// TIA Portal project "FactoryIO_Template_S7-1500_V15_V16" (V16)

(* hardware
DEVICE "S71500/ET200MP-Station_1"  S7-1500 station
   slot 0: "Profilschiene_0"  Rack  6ES7 590-1***0-0AA0
   slot 1: "PLC_1"  CPU 1512C-1 PN  6ES7 512-1CK01-0AB0  V2.8
      slot 3: "CPU-Display_1"  6ES7591-1AA00-0AA0
      slot 32768: "PROFINET-Schnittstelle_1"  X1
         slot 32769: "Port_1"  X1 P1
         slot 32770: "Port_2"  X1 P2
      slot 34817: "Virtual CP interface port_1"  Virtual CP interface port  Virtual CP interface port
   slot 2: "AI 8xU/I/RTD/TC ST_1"  AI 8xU/I/RTD/TC ST  6ES7 531-7KF00-0AB0  V2.0
   slot 3: "AI 8xU/I/RTD/TC ST_2"  AI 8xU/I/RTD/TC ST  6ES7 531-7KF00-0AB0  V2.0
   slot 4: "AI 8xU/I/RTD/TC ST_3"  AI 8xU/I/RTD/TC ST  6ES7 531-7KF00-0AB0  V2.0
   slot 5: "AI 8xU/I/RTD/TC ST_4"  AI 8xU/I/RTD/TC ST  6ES7 531-7KF00-0AB0  V2.0
   slot 6: "DI 16x24VDC BA_1"  DI 16x24VDC BA  6ES7 521-1BH10-0AA0  V1.0
DEVICE "HMI_2"  KTP700 Basic PN
   slot 0: "HMI_2"  KTP700 Basic PN  6AV2 123-2GB03-0AX0  16.0.0.0
   slot 1: "HMI_RT_2"  KTP700 Basic PN  6AV2 123-2GB03-0AX0  16.0.0.0
   slot 5: "HMI_2.IE_CP_1"  PROFINET Interface  16.0.0.0
      slot 1: "PROFINET Interface_1"  PROFINET Interface
         slot 1: "Port_1"  Port
*)

// ===== PLC "PLC_1"  CPU 1512C-1 PN =====

VAR_GLOBAL   // PLC tag table "Standard-Variablentabelle"
   "Tag_1" AT %M0.1 : Bool;
   "Tag_2" AT %M0.0 : Bool;
END_VAR

VAR_GLOBAL   // PLC tag table "Inputs"
   "Flow_Rate_Sensor" AT %I1.0 : Bool;
   "Float_switch_overflow" AT %I1.1 : Bool;   // S111
   "Float_switch_threshold" AT %I1.2 : Bool;   // S112
   "Low_Level_Capacitive_Sensor" AT %I1.3 : Bool;   // B114
   "High_Level_Capacitive_Sensor" AT %I1.4 : Bool;   // B113
   "Micro_switch_valve_closed" AT %I1.5 : Bool;
   "Micro_switch_valve_open" AT %I1.6 : Bool;
   "Ultrasonic_Sensor" AT %IW96 : Int;
END_VAR

VAR_GLOBAL   // PLC tag table "Outputs"
   "Solenoid_on/off" AT %Q1.0 : Bool;
   "Heater_on/off" AT %Q1.1 : Bool;
   "Relay KF1_Pump mode" AT %Q1.2 : Bool;
   "Pump_on/off" AT %Q1.3 : Bool;
   "KF6_Proportional valve" AT %Q1.4 : Bool;
   "KF2_Fan" AT %Q1.5 : Bool;
   "Pump_P101" AT %QW96 : Int;
END_VAR

VAR_GLOBAL   // PLC tag table "Factory tags"
   "FactoryIO_running" AT %I0.3 : Bool;
   "Ultrasonic_Sensor_factory" AT %ID30 : Real;
   "Fill valve" AT %QD30 : Real;
   "Discharge valve" AT %QD34 : Real;
   "SP" AT %QD38 : DInt;
   "Flow meter" AT %ID34 : Real;
   "setpoint" AT %ID38 : Real;
   "PV" AT %QD42 : DInt;
   "Start" AT %I0.0 : Bool;
   "Reset" AT %I0.1 : Bool;
   "Stop" AT %I0.2 : Bool;
   "Start light" AT %Q0.0 : Bool;
   "Reset light" AT %Q0.1 : Bool;
   "Stop light" AT %Q0.2 : Bool;
END_VAR

// folder: Sys_par

DATA_BLOCK "sys_utils"   // DB3
{ S7_Optimized_Access := 'TRUE' }
VERSION : 0.1
   VAR
      "toggle tags" : Bool;
      process_type : Int := 0;
      _xState_pump : Bool;
      _xState_discharge : Bool;
      _xState_Start : Bool;
      _xState_Reset : Bool;
      _xState_Stop : Bool;
      _xState_PIDState : Bool;
   END_VAR
BEGIN
END_DATA_BLOCK

DATA_BLOCK "parameters"   // DB4
{ S7_Optimized_Access := 'TRUE' }
VERSION : 0.1
   VAR
      "Process Value" : Real;
      setpoint : DInt := 0;
      setpoint_pid : Real;
      flowrate : Real;
      ModeActivate : Bool;
      ManualEnable : Bool;
      InactiveEnable : Bool;
      ManualValue : Real := 80.0;
      Inactive : Int := 0;
      Reset : Bool;
      "Error_Discharge valve" : Real;
      "Flow_Meter buffer" : Real;
      "Level Buffer" : Real;
      "Setpoint buffer" : Real;
      Error : Real;
      PWM_DISABLE : Bool;
   END_VAR
BEGIN
END_DATA_BLOCK

// folder: (top level)

FUNCTION "Control_Unit" : Void   // FC1, LAD
{ S7_Optimized_Access := 'TRUE' }
VERSION : 0.1
   VAR_TEMP
      stop_light : Bool;
      start_light : Bool;
   END_VAR
   VAR_TEMP   // added for the SCL form of the ladder/FBD networks
      _w1 : Bool;
      _w2 : Bool;
   END_VAR
BEGIN

REGION Network 1: Stop condition
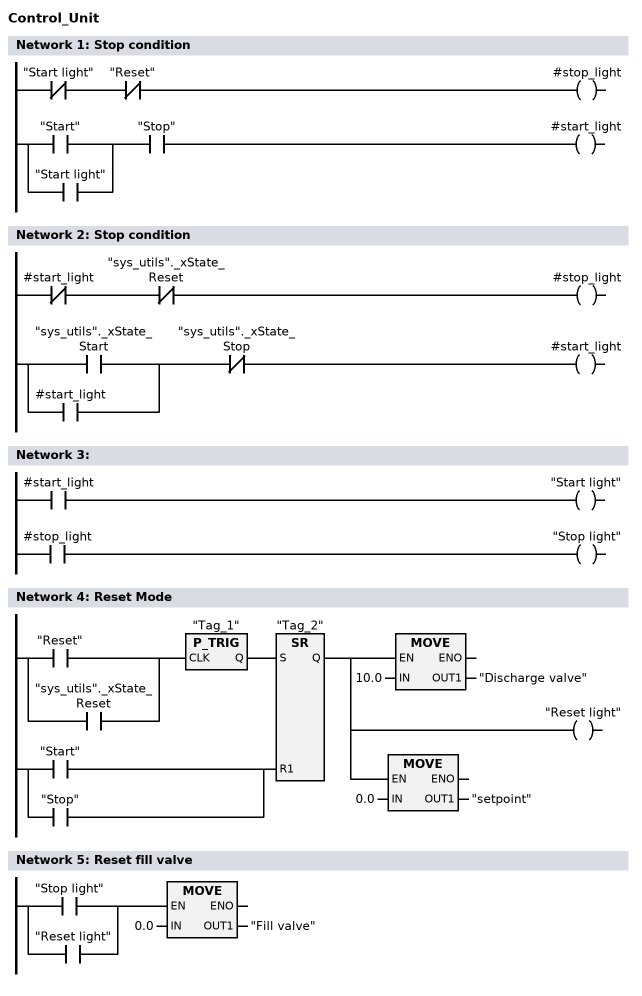
   RUNG wire#powerrail
      I_Contact( "Start light" )
      I_Contact( "Reset" )
      Coil( #stop_light )
   END_RUNG
   RUNG wire#powerrail
      Contact( "Start" )
      wire#w1
      Contact( "Stop" )
      Coil( #start_light )
   END_RUNG
   RUNG wire#powerrail
      Contact( "Start light" )
   END_RUNG wire#w1
   // the same network as SCL:
   #stop_light := NOT "Start light" AND NOT "Reset";
   #start_light := ("Start" OR "Start light") AND "Stop";
END_REGION

REGION Network 2: Stop condition
   RUNG wire#powerrail
      I_Contact( #start_light )
      I_Contact( "sys_utils"._xState_Reset )
      Coil( #stop_light )
   END_RUNG
   RUNG wire#powerrail
      Contact( "sys_utils"._xState_Start )
      wire#w1
      I_Contact( "sys_utils"._xState_Stop )
      Coil( #start_light )
   END_RUNG
   RUNG wire#powerrail
      Contact( #start_light )
   END_RUNG wire#w1
   // the same network as SCL:
   #stop_light := NOT #start_light AND NOT "sys_utils"._xState_Reset;
   #start_light := ("sys_utils"._xState_Start OR #start_light) AND NOT "sys_utils"._xState_Stop;
END_REGION

REGION Network 3
   RUNG wire#powerrail
      Contact( #start_light )
      Coil( "Start light" )
   END_RUNG
   RUNG wire#powerrail
      Contact( #stop_light )
      Coil( "Stop light" )
   END_RUNG
   // the same network as SCL:
   "Start light" := #start_light;
   "Stop light" := #stop_light;
END_REGION

REGION Network 4: Reset Mode
   RUNG wire#powerrail
      Contact( "Reset" )
      wire#w1
      P_Trig( "Tag_1" )
      S_SR(operand := "Tag_2", r1 := wire#w2)
      wire#w3
      Move(in := 10.0, out1 => "Discharge valve")
   END_RUNG
   RUNG wire#powerrail
      Contact( "sys_utils"._xState_Reset )
   END_RUNG wire#w1
   RUNG wire#powerrail
      Contact( "Start" )
   END_RUNG wire#w2
   RUNG wire#powerrail
      Contact( "Stop" )
   END_RUNG wire#w2
   RUNG wire#w3
      Coil( "Reset light" )
   END_RUNG
   RUNG wire#w3
      Move(in := 0.0, out1 => "setpoint")
   END_RUNG
   // the same network as SCL:
   #_w1 := "Reset" OR "sys_utils"._xState_Reset;
   #_w2 := #_w1 AND NOT "Tag_1";   // rising edge
   "Tag_1" := #_w1;
   IF #_w2 THEN
       "Tag_2" := TRUE;   // SR flip-flop
   END_IF;
   IF "Start" OR "Stop" THEN "Tag_2" := FALSE; END_IF;
   IF "Tag_2" THEN "Discharge valve" := 10.0; END_IF;
   "Reset light" := "Tag_2";
   IF "Tag_2" THEN "setpoint" := 0.0; END_IF;
END_REGION

REGION Network 5: Reset fill valve
   RUNG wire#powerrail
      Contact( "Stop light" )
      wire#w1
      Move(in := 0.0, out1 => "Fill valve")
   END_RUNG
   RUNG wire#powerrail
      Contact( "Reset light" )
   END_RUNG wire#w1
   // the same network as SCL:
   IF "Stop light" OR "Reset light" THEN "Fill valve" := 0.0; END_IF;
END_REGION
END_FUNCTION

FUNCTION "height_conversion" : Void   // FC3, LAD
{ S7_Optimized_Access := 'TRUE' }
VERSION : 0.1
   VAR_INPUT
      height_sensor : Real;
   END_VAR
   VAR_OUTPUT
      scaled_height : DInt;
   END_VAR
   VAR_TEMP
      norm_height : Real;
   END_VAR
BEGIN

REGION Network 1: Height Conversion
   // 1. Normalize the sensor output data between 0.0 and 1.0
   // 2. Scale the normalized data between minimum and maximum scale reading
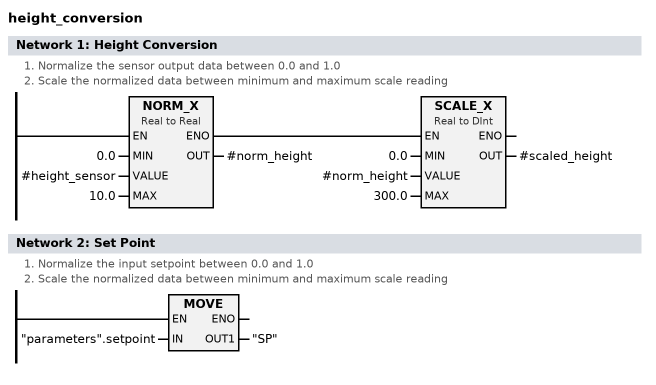
   RUNG wire#powerrail
      { S7_Templates := "[SrcType := Real, DestType := Real]" } Normalize(min := 0.0, value := #height_sensor, max := 10.0, out => #norm_height)
      { S7_Templates := "[SrcType := Real, DestType := DInt]" } Scale(min := 0.0, value := #norm_height, max := 300.0, out => #scaled_height)
   END_RUNG
   // the same network as SCL:
   #norm_height := NORM_X(MIN := 0.0, VALUE := #height_sensor, MAX := 10.0);
   #scaled_height := SCALE_X(MIN := 0.0, VALUE := #norm_height, MAX := 300.0);
END_REGION

REGION Network 2: Set Point
   // 1. Normalize the input setpoint between 0.0 and 1.0
   // 2. Scale the normalized data between minimum and maximum scale reading
   RUNG wire#powerrail
      Move(in := "parameters".setpoint, out1 => "SP")
   END_RUNG
   // the same network as SCL:
   "SP" := "parameters".setpoint;
END_REGION
END_FUNCTION

FUNCTION "MHJ-PLC-Lab-Function-S71500" : Void   // FC9000, SCL
{ S7_Optimized_Access := 'TRUE' }
VERSION : 0.1
   VAR_TEMP
      Value : Byte;
      ForCounter : Int;
   END_VAR
   VAR CONSTANT
      Value_01_DW : DWord := 16#1223_5486;
      Value_02_DW : DWord := 16#A6C9_D1F5;
   END_VAR
BEGIN

   #Value:=PEEK(area := 16#82,
        dbNumber := 0,
        byteOffset := 511);
   #Value := #Value + 1;

   POKE(area := 16#82,
        dbNumber := 0,
        byteOffset := 511,
        value := #Value);

   POKE(area := 16#82,
        dbNumber := 0,
        byteOffset := 1016,
        value := #Value_01_DW);
   POKE(area := 16#82,
        dbNumber := 0,
        byteOffset := 1020,
        value := #Value_02_DW);

   FOR #ForCounter := 0 TO 63 DO
       #Value:=PEEK(area := 16#1,
            dbNumber := 0,
            byteOffset := #ForCounter);
       POKE(area := 16#81,
            dbNumber := 0,
            byteOffset := #ForCounter,
            value := #Value);
   END_FOR;
   #Value := PEEK(area := 16#1,
                  dbNumber := 0,
                  byteOffset := 512);
   POKE(area := 16#82,
        dbNumber := 0,
        byteOffset := 512,
        value := #Value);
END_FUNCTION

ORGANIZATION_BLOCK "Main"   // OB1, LAD, ProgramCycle
TITLE = "Main Program Sweep (Cycle)"
{ S7_Optimized_Access := 'TRUE' }
VERSION : 0.1
   VAR_INPUT
      Initial_Call : Bool;   // Initial call of this OB
      Remanence : Bool;   // =True, if remanent data are available
   END_VAR
BEGIN

REGION Network 1
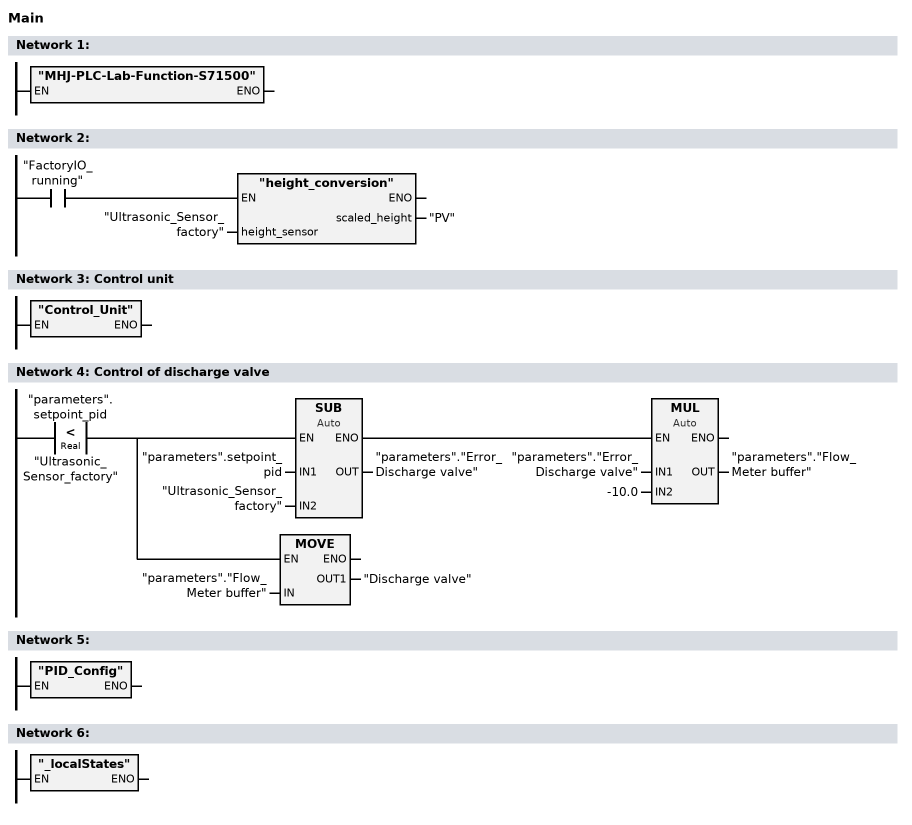
   RUNG wire#powerrail
      "MHJ-PLC-Lab-Function-S71500"()
   END_RUNG
   // the same network as SCL:
   "MHJ-PLC-Lab-Function-S71500"();
END_REGION

REGION Network 2
   RUNG wire#powerrail
      Contact( "FactoryIO_running" )
      "height_conversion"(height_sensor := "Ultrasonic_Sensor_factory", scaled_height => "PV")
   END_RUNG
   // the same network as SCL:
   IF "FactoryIO_running" THEN
       "height_conversion"(height_sensor := "Ultrasonic_Sensor_factory", scaled_height => "PV");
   END_IF;
END_REGION

REGION Network 3: Control unit
   RUNG wire#powerrail
      "Control_Unit"()
   END_RUNG
   // the same network as SCL:
   "Control_Unit"();
END_REGION

REGION Network 4: Control of discharge valve
   RUNG wire#powerrail
      { S7_Templates := "SrcType := Real" } LT_Contact(in1 := "parameters".setpoint_pid, in2 := "Ultrasonic_Sensor_factory")
      wire#w1
      Sub(in1 := "parameters".setpoint_pid, in2 := "Ultrasonic_Sensor_factory", out => "parameters"."Error_Discharge valve")
      Mul(in1 := "parameters"."Error_Discharge valve", in2 := -10.0, out => "parameters"."Flow_Meter buffer")
   END_RUNG
   RUNG wire#w1
      Move(in := "parameters"."Flow_Meter buffer", out1 => "Discharge valve")
   END_RUNG
   // the same network as SCL:
   IF "parameters".setpoint_pid < "Ultrasonic_Sensor_factory" THEN
       "parameters"."Error_Discharge valve" := "parameters".setpoint_pid - "Ultrasonic_Sensor_factory";
       "parameters"."Flow_Meter buffer" := "parameters"."Error_Discharge valve" * (-10.0);
       "Discharge valve" := "parameters"."Flow_Meter buffer";
   END_IF;
END_REGION

REGION Network 5
   RUNG wire#powerrail
      "PID_Config"()
   END_RUNG
   // the same network as SCL:
   "PID_Config"();
END_REGION

REGION Network 6
   RUNG wire#powerrail
      "_localStates"()
   END_RUNG
   // the same network as SCL:
   "_localStates"();
END_REGION
END_ORGANIZATION_BLOCK

ORGANIZATION_BLOCK "Cyclic interrupt PID"   // OB30, LAD, CyclicInterrupt
{ S7_Optimized_Access := 'TRUE' }
VERSION : 0.1
   VAR_INPUT
      Initial_Call : Bool;   // Initial call of this OB
      Event_Count : Int;   // Events discarded
   END_VAR
BEGIN

REGION Network 1
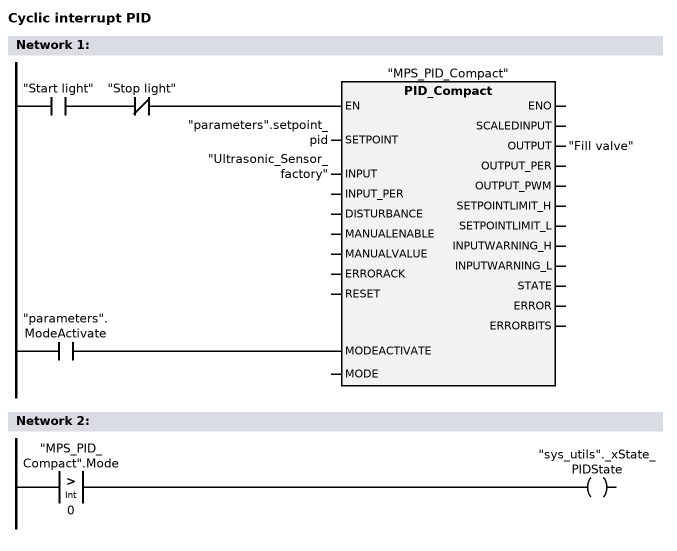
   IF "Start light" AND NOT "Stop light" THEN
       "MPS_PID_Compact"(Setpoint := "parameters".setpoint_pid,   // PID_Compact
                         Input := "Ultrasonic_Sensor_factory",
                         ModeActivate := "parameters".ModeActivate,
                         Output => "Fill valve");
   END_IF;
END_REGION

REGION Network 2
   RUNG wire#powerrail
      { S7_Templates := "SrcType := Int" } GT_Contact(in1 := "MPS_PID_Compact".Mode, in2 := 0)
      Coil( "sys_utils"._xState_PIDState )
   END_RUNG
   // the same network as SCL:
   "sys_utils"._xState_PIDState := "MPS_PID_Compact".Mode > 0;
END_REGION
END_ORGANIZATION_BLOCK

// folder: Sys_par

FUNCTION "PID_Config" : Void   // FC2, LAD
{ S7_Optimized_Access := 'TRUE' }
VERSION : 0.1
   VAR_TEMP
      norm_setpoint : Real;
   END_VAR
BEGIN

REGION Network 1: enable mode
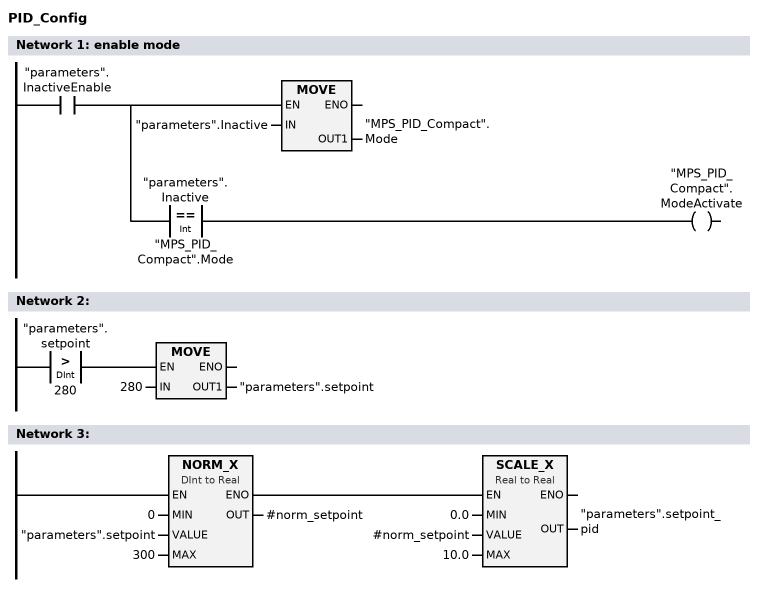
   RUNG wire#powerrail
      Contact( "parameters".InactiveEnable )
      wire#w1
      Move(in := "parameters".Inactive, out1 => "MPS_PID_Compact".Mode)
   END_RUNG
   RUNG wire#w1
      { S7_Templates := "SrcType := Int" } EQ_Contact(in1 := "parameters".Inactive, in2 := "MPS_PID_Compact".Mode)
      Coil( "MPS_PID_Compact".ModeActivate )
   END_RUNG
   // the same network as SCL:
   IF "parameters".InactiveEnable THEN "MPS_PID_Compact".Mode := "parameters".Inactive; END_IF;
   "MPS_PID_Compact".ModeActivate := "parameters".InactiveEnable AND ("parameters".Inactive = "MPS_PID_Compact".Mode);
END_REGION

REGION Network 2
   RUNG wire#powerrail
      { S7_Templates := "SrcType := DInt" } GT_Contact(in1 := "parameters".setpoint, in2 := 280)
      Move(in := 280, out1 => "parameters".setpoint)
   END_RUNG
   // the same network as SCL:
   IF "parameters".setpoint > 280 THEN "parameters".setpoint := 280; END_IF;
END_REGION

REGION Network 3
   RUNG wire#powerrail
      { S7_Templates := "[SrcType := DInt, DestType := Real]" } Normalize(min := 0, value := "parameters".setpoint, max := 300, out => #norm_setpoint)
      { S7_Templates := "[SrcType := Real, DestType := Real]" } Scale(min := 0.0, value := #norm_setpoint, max := 10.0, out => "parameters".setpoint_pid)
   END_RUNG
   // the same network as SCL:
   #norm_setpoint := NORM_X(MIN := 0, VALUE := "parameters".setpoint, MAX := 300);
   "parameters".setpoint_pid := SCALE_X(MIN := 0.0, VALUE := #norm_setpoint, MAX := 10.0);
END_REGION
END_FUNCTION

FUNCTION "_localStates" : Void   // FC4, LAD
{ S7_Optimized_Access := 'TRUE' }
VERSION : 0.1
BEGIN

REGION Network 1: Pump state
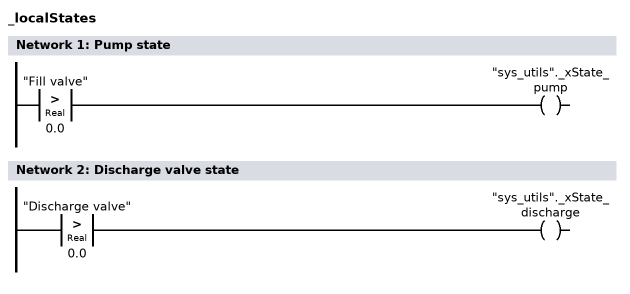
   RUNG wire#powerrail
      { S7_Templates := "SrcType := Real" } GT_Contact(in1 := "Fill valve", in2 := 0.0)
      Coil( "sys_utils"._xState_pump )
   END_RUNG
   // the same network as SCL:
   "sys_utils"._xState_pump := "Fill valve" > 0.0;
END_REGION

REGION Network 2: Discharge valve state
   RUNG wire#powerrail
      { S7_Templates := "SrcType := Real" } GT_Contact(in1 := "Discharge valve", in2 := 0.0)
      Coil( "sys_utils"._xState_discharge )
   END_RUNG
   // the same network as SCL:
   "sys_utils"._xState_discharge := "Discharge valve" > 0.0;
END_REGION
END_FUNCTION

(* ===== HMI "HMI_RT_2" =====
system functions are stored by id; their names below are inferred from use
connection "HMI_Connection_2": ETHERNET, SMART_S7_1500_OMS

HMI tags "Default tag table"
   "Tag_ScreenNumber" : UInt, internal
   "PV" : DInt = PLC PV AT %QD42, 1 s
   "SP" : DInt = PLC SP AT %QD38, 1 s
   "MPS_PID_Compact_CtrlParamsBackUp_Gain" : Real = PLC MPS_PID_Compact.CtrlParamsBackUp.Gain, 1 s
   "MPS_PID_Compact_CtrlParamsBackUp_Ti" : Real = PLC MPS_PID_Compact.CtrlParamsBackUp.Ti, 1 s
   "MPS_PID_Compact_CtrlParamsBackUp_Td" : Real = PLC MPS_PID_Compact.CtrlParamsBackUp.Td, 1 s
   "setpoint" : Real = PLC setpoint AT %ID38, 1 s
   "Start" : Bool = PLC Start AT %I0.0, 1 s
   "Start light" : Bool = PLC "Start light" AT %Q0.0, 1 s
   "Stop" : Bool = PLC Stop AT %I0.2, 1 s
   "Stop light" : Bool = PLC "Stop light" AT %Q0.2, 1 s
   "MPS_PID_Compact_Mode" : Int = PLC MPS_PID_Compact.Mode, 1 s
   "MPS_PID_Compact_ModeActivate" : Bool = PLC MPS_PID_Compact.ModeActivate, 1 s
   "parameters_InactiveEnable" : Bool = PLC parameters.InactiveEnable, 1 s
   "parameters_setpoint" : DInt = PLC parameters.setpoint, 1 s
   "sys_utils_toggle tags" : Bool = PLC sys_utils."toggle tags", 1 s
   "Reset" : Bool = PLC Reset AT %I0.1, 1 s
   "Reset light" : Bool = PLC "Reset light" AT %Q0.1, 1 s
   "sys_utils_process_type" : Int = PLC sys_utils.process_type, 1 s
   "sys_utils__xState_discharge" : Bool = PLC sys_utils._xState_discharge, 1 s
   "sys_utils__xState_pump" : Bool = PLC sys_utils._xState_pump, 1 s
   "sys_utils__xState_Start" : Bool = PLC sys_utils._xState_Start, 1 s
   "sys_utils__xState_Stop" : Bool = PLC sys_utils._xState_Stop, 1 s
   "parameters_ModeActivate" : Bool = PLC parameters.ModeActivate, 1 s
   "sys_utils__xState_Reset" : Bool = PLC sys_utils._xState_Reset, 1 s
   "sys_utils__xState_PIDState" : Bool = PLC sys_utils._xState_PIDState, 1 s

HMI tags "Local Template"
   "_iScreenNumber" : Int, internal
   "_xState_Btn_Overview" : Bool, internal
   "_xState_Btn_Alarm" : Bool, internal
   "_xState_Btn_Recipe" : Bool, internal
   "_xState_Btn_Settings" : Bool, internal
   "_xState_Btn_Level_Overview" : Bool, internal
   "_xState_Btn_Level_Config" : Bool, internal
   "_xState_Btn_Alarm_Buffer" : Bool, internal
   "_xState_Btn_ToggleTags" : Bool, internal
   "_sUserName" : WString[254], internal
   "_iUserGroupNumber" : Int, internal

text list "Text_list_Modes": 3 'Automatic'; 4 'Manual'

text list "Text_list_ToggleTags": 0 'Tags'; 1 'Name'

text list "Text_list_ProcessNames": 1 'Level Control'; 2 'Flow Control'; 3 'Temperature'; 4 'Pressure'; 0 'Home'

graphic list "GraphList_Btn_Template_Settings": 0 'Graphic_13'; 1 'Graphic_12'

graphic list "GraphList_Proportional_Valve": 0 'Graphic_45'; 1 'Graphic_46'

graphic list "GraphList_Pump": 0 'Graphic_27'; 1 'Graphic_26'

graphic list "GraphList_Btn_Template_Recipe": 0 'Graphic_14'; 1 'Graphic_15'

graphic list "GraphList_Btn_Template_Alarm": 0 'Graphic_16'; 1 'Graphic_17'

graphic list "GraphList_Btn_Template_Overview": 0 'Graphic_19'; 1 'Graphic_18'

screen "Alarm" 800x480, template "Template_overview"
   on GenerateScreen: SetBit("_xState_Btn_Alarm"); SetTag("_iScreenNumber", 10)
   on ClearScreen: ResetBit("_xState_Btn_Alarm")
   AlarmView "Alarm view_1" at 5,48 size 592x422
   Button "Template_Button_4" at 600,409 size 83x58; TextOff 'Text'; PictureList "GraphList_Btn_Template_Settings"; PictureOff "Graphic_49"; PictureOn "Graphic_50"; Authorization "Operation"
      ProcessValue <- "_xState_Btn_Settings"
   Button "Template_Button_1" at 600,48 size 83x58; TextOff 'Text'; PictureList "GraphList_Btn_Template_Settings"; PictureOff "Graphic_54"; PictureOn "Graphic_50"
      on Release: ActivateScreen("Alarm Buffer", 0)
      ProcessValue <- "_xState_Btn_Settings"

screen "Level Config" 800x480, template "Template"
   on GenerateScreen: SetBit("_xState_Btn_Level_Config"); SetTag("_iScreenNumber", 2)
   on ClearScreen: ResetBit("_xState_Btn_Level_Config")
   TrendView "Trend view_1" at 38,167 size 644x300
   IOField "I/O field_1" at 442,76 size 105x27; FormatPattern 999.99
      ProcessValue <- "MPS_PID_Compact_CtrlParamsBackUp_Gain"
   IOField "I/O field_2" at 442,105 size 105x27; FormatPattern 99.99
      ProcessValue <- "MPS_PID_Compact_CtrlParamsBackUp_Ti"
   IOField "I/O field_3" at 442,135 size 105x27; FormatPattern 99.99
      ProcessValue <- "MPS_PID_Compact_CtrlParamsBackUp_Td"
   TextField "Text field_1" at 553,80 size 107x23; Text 'Proportional'
   TextField "Text field_2" at 552,108 size 71x23; Text 'Integral'
   TextField "Text field_3" at 552,136 size 89x23; Text 'Derivative'
   Button "Button_1" at 442,47 size 218x28; TextOff 'Save PID Parameters'
   Button "Button_2" at 200,53 size 96x30; TextOff 'Enable'
      on Press: SetBit("parameters_ModeActivate")
      on Release: ResetBit("parameters_ModeActivate")
      Appearance <- "sys_utils__xState_PIDState"
   Button "Button_5" at 305,53 size 96x31; TextOff 'Disable'
      on Release: ResetBit("parameters_InactiveEnable")
      on Press: SetBit("parameters_InactiveEnable")
   IOField "I/O field_4" at 43,129 size 105x33; FormatPattern 999
      ProcessValue <- "parameters_setpoint"
   TextField "Text field_4" at 43,106 size 75x23; Text 'SetPoint'
   IOField "I/O field_5" at 278,126 size 105x33; FormatPattern 999
      ProcessValue <- "PV"
   TextField "Text field_5" at 272,105 size 118x23; Text 'Process Value'
   SymbolicIOField "Symbolic I/O field_1" at 38,51 size 159x32; TextOff '0'; TextOn '1'; TextList "Text_list_Modes"
      ProcessValue <- "MPS_PID_Compact_Mode"
   Button "Button_3" at 157,0 size 160x40; TextOff 'OverView'
      Appearance <- "_xState_Btn_Level_Overview"
      on Release: ActivateScreen("Level OverView", 0); SetBit("_xState_Btn_Level_Overview"); ResetBit("_xState_Btn_Level_Config")
   Button "Button_4" at 322,1 size 145x40; TextOff 'Configuration'
      on Release: ActivateScreen("Level Config", 0); SetBit("_xState_Btn_Level_Config"); ResetBit("_xState_Btn_Level_Overview")
      Appearance <- "_xState_Btn_Level_Config"

screen "Level OverView" 800x480, template "Template"
   on GenerateScreen: SetBit("_xState_Btn_Level_Overview"); SetTag("_iScreenNumber", 2)
   on ClearScreen: ResetBit("_xState_Btn_Level_Overview")
   GraphicView "Graphic view_4" at 128,89 size 150x187; Picture "Graphic_25"
   GraphicView "Graphic view_1" at 416,163 size 148x178; Picture "Graphic_25"
   Circle "Circle_5" at 393,433 size 25x25
      Appearance <- "sys_utils__xState_PIDState"
   GraphicView "Graphic view_21" at 319,78 size 45x23; Picture "Graphic_40"
   GraphicView "Graphic view_25" at 222,281 size 40x21; Picture "Graphic_40"
   GraphicView "Graphic view_18" at 85,270 size 31x44; Picture "Graphic_39"
   GraphicView "Graphic view_20" at 502,367 size 51x31; Picture "Graphic_40"
   Bar "Bar_1" at 140,124 size 128x115; MinimumValue 0; MaximumValue 300
      ProcessValue <- "PV"
   Button "Button_3" at 157,0 size 160x40; TextOff 'OverView'
      on Release: ActivateScreen("Level OverView", 0); SetBit("_xState_Btn_Level_Overview"); ResetBit("_xState_Btn_Level_Config")
      Appearance <- "_xState_Btn_Level_Overview"
   Button "Button_4" at 322,1 size 145x40; TextOff 'Configuration'
      on Release: ActivateScreen("Level Config", 0); SetBit("_xState_Btn_Level_Config"); ResetBit("_xState_Btn_Level_Overview")
      Appearance <- "_xState_Btn_Level_Config"
   Button "Button_1" at 432,372 size 43x52; TextOff 'Text'; PictureList "GraphList_Pump"
      ProcessValue <- "sys_utils__xState_pump"
   GraphicView "Graphic view_2" at 116,382 size 322x34; Picture "Graphic_28"
   GraphicView "Graphic view_7" at 81,383 size 36x32; Picture "Graphic_32"
   GraphicView "Graphic view_3" at 83,310 size 34x75; Picture "Graphic_33"
   GraphicView "Graphic view_5" at 111,211 size 30x34; Picture "Graphic_28"
   GraphicView "Graphic view_6" at 474,333 size 34x38; Picture "Graphic_33"
   GraphicView "Graphic view_8" at 474,363 size 35x41; Picture "Graphic_36"
   GraphicView "Graphic view_9" at 191,258 size 34x22; Picture "Graphic_33"
   GraphicView "Graphic view_10" at 259,275 size 173x34; Picture "Graphic_28"
   GraphicView "Graphic view_11" at 266,116 size 27x34; Picture "Graphic_28"
   GraphicView "Graphic view_12" at 357,71 size 137x34; Picture "Graphic_28"
   GraphicView "Graphic view_13" at 524,71 size 83x34; Picture "Graphic_28"
   GraphicView "Graphic view_14" at 547,187 size 59x34; Picture "Graphic_28"
   GraphicView "Graphic view_15" at 604,98 size 34x94; Picture "Graphic_33"
   GraphicView "Graphic view_16" at 194,60 size 31x41; Picture "Graphic_37"
   GraphicView "Graphic view_17" at 190,276 size 36x32; Picture "Graphic_32"
   GraphicView "Graphic view_19" at 290,114 size 37x37; Picture "Graphic_42"
   GraphicView "Graphic view_23" at 291,104 size 34x16; Picture "Graphic_33"
   GraphicView "Graphic view_24" at 292,75 size 33x31; Picture "Graphic_43"
   GraphicView "Graphic view_26" at 84,212 size 33x33; Picture "Graphic_43"
   GraphicView "Graphic view_27" at 83,241 size 34x38; Picture "Graphic_33"
   GraphicView "Graphic view_28" at 544,366 size 30x34; Picture "Graphic_28"
   GraphicView "Graphic view_29" at 602,186 size 37x37; Picture "Graphic_42"
   GraphicView "Graphic view_30" at 603,70 size 37x37; Picture "Graphic_44"
   Button "Button_2" at 491,67 size 36x41; TextOff 'Text'; PictureList "GraphList_Proportional_Valve"
      ProcessValue <- "sys_utils__xState_discharge"
   GraphicView "Graphic view_31" at 560,343 size 82x83; Picture "Graphic_48"
   TextField "Text field_1" at 58,187 size 45x23; Text 'S112'
      Visibility <- "_xState_Btn_ToggleTags"
   TextField "Text field_2" at 224,50 size 46x23; Text 'B102'
      Visibility <- "_xState_Btn_ToggleTags"
   TextField "Text field_3" at 340,186 size 46x23; Text 'B113'
      Visibility <- "_xState_Btn_ToggleTags"
   TextField "Text field_4" at 594,287 size 46x23; Text 'B114'
      Visibility <- "_xState_Btn_ToggleTags"
   TextField "Text field_5" at 424,140 size 45x23; Text 'S111'
      Visibility <- "_xState_Btn_ToggleTags"
   TextField "Text field_6" at 466,48 size 113x20; Text 'Proportion valve'
      Visibility <- "_xState_Btn_ToggleTags"
   TextField "Text field_7" at 120,287 size 46x23; Text 'V101'
      Visibility <- "_xState_Btn_ToggleTags"
   TextField "Text field_8" at 221,302 size 46x23; Text 'V110'
      Visibility <- "_xState_Btn_ToggleTags"
   TextField "Text field_9" at 504,396 size 46x23; Text 'V105'
      Visibility <- "_xState_Btn_ToggleTags"
   TextField "Text field_10" at 319,103 size 46x23; Text 'V112'
      Visibility <- "_xState_Btn_ToggleTags"
   TextField "Text field_11" at 508,142 size 82x20; Text 'Float switch'
      Visibility <- "_xState_Btn_ToggleTags"
   TextField "Text field_12" at 580,266 size 101x20; Text 'Low Level Cap.'
      Visibility <- "_xState_Btn_ToggleTags"
   TextField "Text field_13" at 288,165 size 103x20; Text 'High Level Cap.'
      Visibility <- "_xState_Btn_ToggleTags"
   TextField "Text field_14" at 56,162 size 82x20; Text 'Float switch'
      Visibility <- "_xState_Btn_ToggleTags"
   TextField "Text field_15" at 224,68 size 69x20; Text 'Ultrasonic'
      Visibility <- "_xState_Btn_ToggleTags"
   TextField "Text field_16" at 344,415 size 49x26; Text 'PID'
   SymbolicIOField "Symbolic I/O field_1" at 694,198 size 97x32; TextOff '0'; TextOn '1'; TextList "Text_list_ToggleTags"
      ProcessValue <- "_xState_Btn_ToggleTags"
   TextField "Text field_17" at 404,346 size 49x26; Text 'Pump'
      Visibility <- "_xState_Btn_ToggleTags"
   Line "Line_6" at 387,398 size 51x0
      Appearance <- "sys_utils__xState_pump"
      Visibility <- "sys_utils__xState_pump"
   Line "Line_7" at 261,291 size 51x0
      Appearance <- "sys_utils__xState_discharge"
      Visibility <- "sys_utils__xState_discharge"

screen "Alarm Buffer" 800x480, template "Template_overview"
   on GenerateScreen: SetBit("_xState_Btn_Alarm"); SetTag("_iScreenNumber", 10)
   on ClearScreen: ResetBit("_xState_Btn_Alarm_Buffer")
   AlarmView "Alarm view_1" at 5,48 size 592x422
   Button "Template_Button_4" at 600,49 size 83x58; TextOff 'Text'; PictureList "GraphList_Btn_Template_Settings"; PictureOff "Graphic_52"; PictureOn "Graphic_50"
      on Release: function_efd93a16()
      ProcessValue <- "_xState_Btn_Settings"

screen "Recipe" 800x480, template "Template_overview"
   on GenerateScreen: SetBit("_xState_Btn_Recipe"); SetTag("_iScreenNumber", 15)
   on ClearScreen: ResetBit("_xState_Btn_Recipe")

screen "Overview" 800x480, template "Template_overview"
   on GenerateScreen: SetBit("_xState_Btn_Overview"); SetTag("_iScreenNumber", 1)
   on ClearScreen: ResetBit("_xState_Btn_Overview")
   Button "Button_1" at 140,201 size 182x58; TextOff 'Level Control'; PictureOff "level_ind"
      on Release: ActivateScreen("Level OverView", 0); function_b3f726e6("sys_utils_process_type", 1)
   Button "Button_2" at 377,203 size 183x54; TextOff 'Flow Control'; PictureOff "level_ind"
      on Release: function_b3f726e6("sys_utils_process_type", 2)
   Button "Button_3" at 143,284 size 182x58; TextOff 'Temperature'; PictureOff "level_ind"
      on Release: function_b3f726e6("sys_utils_process_type", 3)
   Button "Button_4" at 377,283 size 182x58; TextOff 'Pressure Control'; PictureOff "level_ind"
      on Release: function_b3f726e6("sys_utils_process_type", 4)

screen "Settings" 800x480, template "Template_overview"
   on GenerateScreen: SetBit("_xState_Btn_Settings"); SetTag("_iScreenNumber", 20)
   on ClearScreen: ResetBit("_xState_Btn_Settings")
   Button "Template_Button_1" at 46,84 size 83x58; TextOff 'Text'; PictureList "GraphList_Btn_Template_Settings"; PictureOn "Graphic_50"; PictureOff "Graphic_2"; Authorization "Maintenance"
      ProcessValue <- "_xState_Btn_Settings"
      on Release: function_bc3e350c()
   Button "Template_Button_2" at 203,84 size 83x58; TextOff 'Text'; PictureList "GraphList_Btn_Template_Settings"; PictureOn "Graphic_50"; PictureOff "Graphic_3"; Authorization "Operation"
      ProcessValue <- "_xState_Btn_Settings"
      on Release: function_be740847(15)
   Button "Template_Button_3" at 46,235 size 83x58; TextOff 'Text'; PictureList "GraphList_Btn_Template_Settings"; PictureOn "Graphic_50"; PictureOff "Graphic_6"; Authorization "Operation"
      ProcessValue <- "_xState_Btn_Settings"
      on Release: function_f23ef4c9()
   Button "Template_Button_4" at 205,236 size 83x58; TextOff 'Text'; PictureList "GraphList_Btn_Template_Settings"; PictureOn "Graphic_50"; PictureOff "Graphic_5"; Authorization "Maintenance"
      ProcessValue <- "_xState_Btn_Settings"
      on Release: StopRuntime(0)
   TextField "Text field_14" at 9,143 size 161x39; Text 'CALIBRATE'
      Visibility <- "_xState_Btn_ToggleTags"
   TextField "Text field_1" at 163,144 size 161x39; Text 'CLEAN'
      Visibility <- "_xState_Btn_ToggleTags"
   TextField "Text field_2" at 11,295 size 161x39; Text 'LOG OFF'
      Visibility <- "_xState_Btn_ToggleTags"
   TextField "Text field_3" at 170,296 size 161x39; Text 'EXIT'
      Visibility <- "_xState_Btn_ToggleTags"
   TextField "Text field_13" at 354,56 size 132x20; Text 'Project Information'
      Visibility <- "_xState_Btn_ToggleTags"
   TextField "Text field_4" at 355,84 size 132x37; Text 'Project Information'
      Visibility <- "_xState_Btn_ToggleTags"
   TextField "Text field_5" at 355,119 size 132x37; Text 'Created On'
      Visibility <- "_xState_Btn_ToggleTags"
   TextField "Text field_6" at 356,157 size 132x37; Text 'Author'
      Visibility <- "_xState_Btn_ToggleTags"
   TextField "Text field_7" at 356,195 size 132x37; Text 'Description'
      Visibility <- "_xState_Btn_ToggleTags"
   TextField "Text field_8" at 353,247 size 133x20; Text 'System Information'
      Visibility <- "_xState_Btn_ToggleTags"
   TextField "Text field_9" at 353,278 size 132x37; Text 'PLC DEVICE TYPE:'
      Visibility <- "_xState_Btn_ToggleTags"
   TextField "Text field_10" at 354,315 size 132x37; Text 'HMI DEVICE TYPE:'
      Visibility <- "_xState_Btn_ToggleTags"
   TextField "Text field_11" at 355,352 size 132x37; Text 'CONNECTION TYPE:'
      Visibility <- "_xState_Btn_ToggleTags"
   TextField "Text field_12" at 516,84 size 154x37; Text 'MPS COMPACT FESTO'
      Visibility <- "_xState_Btn_ToggleTags"

Template "Template_overview" 800x480
   Button "Template_Button_1" at 708,43 size 86x75; TextOff 'Text'; PictureList "GraphList_Btn_Template_Overview"
      on Release: ActivateScreen("Overview", 0)
      ProcessValue <- "_xState_Btn_Overview"
   Button "Template_Button_2" at 708,121 size 86x75; TextOff 'Text'; PictureList "GraphList_Btn_Template_Alarm"
      on Release: ActivateScreen("Alarm", 0)
      ProcessValue <- "_xState_Btn_Alarm"
   Button "Template_Button_3" at 708,199 size 86x75; TextOff 'Text'; PictureList "GraphList_Btn_Template_Recipe"
      on Release: ActivateScreen("Recipe", 0)
      ProcessValue <- "_xState_Btn_Recipe"
   Button "Template_Button_4" at 707,277 size 86x75; TextOff 'Text'; PictureList "GraphList_Btn_Template_Settings"
      on Release: ActivateScreen("Settings", 0)
      ProcessValue <- "_xState_Btn_Settings"
   Rectangle "Template_Rectangle_6" at 467,0 size 224x38
      Appearance <- "_iUserGroupNumber"
   Button "Template_Button_5" at 712,415 size 83x58; TextOff 'Text'; PictureList "GraphList_Btn_Template_Settings"; PictureOff "Graphic_52"; PictureOn "Graphic_50"
      on Release: function_efd93a16()
      ProcessValue <- "_xState_Btn_Settings"
   IOField "Template_I/O field_1" at 483,1 size 182x36; FormatPattern ??????????
      ProcessValue <- "_sUserName"
   SymbolicIOField "Template_Symbolic I/O field_1" at 27,4 size 110x32; TextOff '0'; TextOn '1'; TextList "TextList_ScreenNames"
      ProcessValue <- "_iScreenNumber"

Template "Template" 800x480
   Button "Template_Button_2" at 694,40 size 100x75; TextOff 'Text'; PictureList "GraphList_Btn_Template_Alarm"
      on Release: ActivateScreen("Alarm", 0)
      ProcessValue <- "_xState_Btn_Alarm"
   Button "Template_Button_3" at 694,118 size 100x75; TextOff 'Text'; PictureList "GraphList_Btn_Template_Recipe"
      on Release: ActivateScreen("Recipe", 0)
      ProcessValue <- "_xState_Btn_Recipe"
   Button "Template_Button_5" at 695,317 size 82x77; TextOff 'Text'; Authorization "Operation"
      on Release: ResetBit("sys_utils__xState_Stop")
      on Press: SetBit("sys_utils__xState_Stop")
      Appearance <- "Stop light"
   Button "Template_Button_6" at 695,395 size 80x79; TextOff 'Text'; Authorization "Operation"
      on Release: ResetBit("sys_utils__xState_Reset")
      on Press: SetBit("sys_utils__xState_Reset")
      Appearance <- "Reset light"
   Button "Template_Button_4" at 694,238 size 82x77; TextOff 'Text'; Authorization "Operation"
      on Release: ResetBit("sys_utils__xState_Start")
      on Press: SetBit("sys_utils__xState_Start")
   Button "Template_Button_1" at 694,0 size 101x38; TextOff 'Text'; PictureOff "Graphic_18"
      on Release: ActivateScreen("Overview", 0)
   Rectangle "Template_Rectangle_6" at 467,0 size 224x38
      Appearance <- "_iUserGroupNumber"
   IOField "Template_I/O field_1" at 483,1 size 182x36; FormatPattern ??????????
      ProcessValue <- "_sUserName"
   Circle "Template_Circle_1" at 700,319 size 74x74
      Appearance <- "Stop light"
   Circle "Template_Circle_2" at 698,397 size 74x74
      Appearance <- "Reset light"
   Circle "Template_Circle_3" at 698,239 size 74x74
      Appearance <- "Start light"
   TextField "Template_Text field_1" at 774,256 size 24x45; Text 'Start'
   TextField "Template_Text field_2" at 776,334 size 24x41; Text 'Stop'
   TextField "Template_Text field_3" at 774,409 size 24x51; Text 'Reset'
   SymbolicIOField "Template_Symbolic I/O field_1" at 27,4 size 110x32; TextOn '1'; TextOff '0'; TextList "TextList_ScreenNames"
      ProcessValue <- "_iScreenNumber"

scheduled task "UserAdmin"
   on Action: function_f41c6f6c("_sUserName"); function_e1ab61de("_iUserGroupNumber")
*)